// SIMATIC S7-200 project (STEP 7-Micro/WIN), CPU 221 REL 01.10

SYMBOL_TABLE 用户定义1
开1               I0.1
开2               I0.2
关                I0.3
关闭               I0.0
电1               Q0.1
电2               Q0.0
中点               M0.0
END_SYMBOL_TABLE

ORGANIZATION_BLOCK 主程序:OB1
TITLE=程序注释
BEGIN
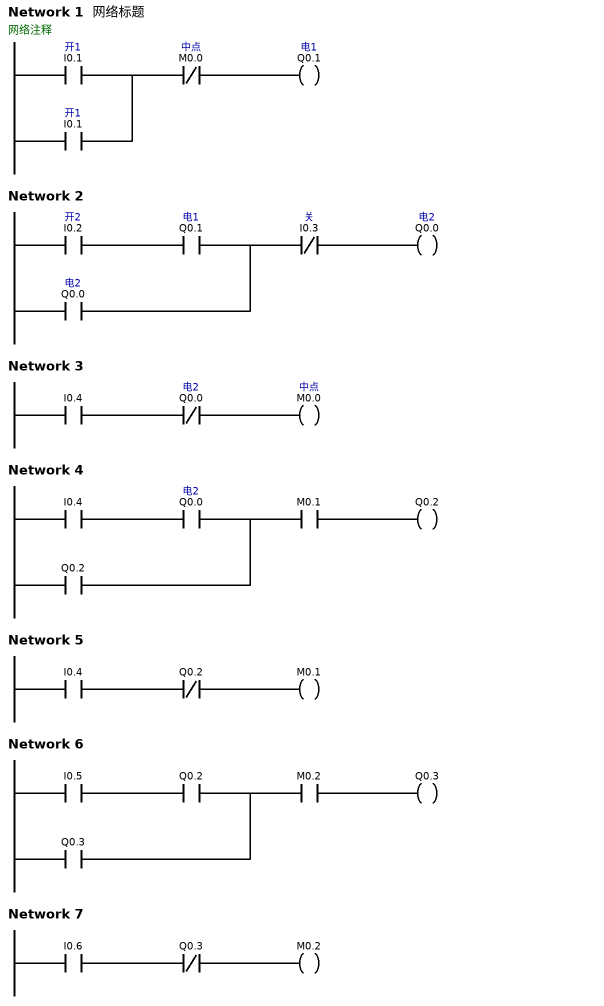
Network 1 // 网络标题
// 网络注释
LD     开1:I0.1
O      开1:I0.1
AN     中点:M0.0
=      电1:Q0.1
Network 2
LD     开2:I0.2
A      电1:Q0.1
O      电2:Q0.0
AN     关:I0.3
=      电2:Q0.0
Network 3
LD     I0.4
AN     电2:Q0.0
=      中点:M0.0
Network 4
LD     I0.4
A      电2:Q0.0
O      Q0.2
A      M0.1
=      Q0.2
Network 5
LD     I0.4
AN     Q0.2
=      M0.1
Network 6
LD     I0.5
A      Q0.2
O      Q0.3
A      M0.2
=      Q0.3
Network 7
LD     I0.6
AN     Q0.3
=      M0.2
END_ORGANIZATION_BLOCK
